PROGRAM P_Composite
VAR
	machine01				: Machine;
END_VAR

machine01.logStatus();

END_PROGRAM

(* stored: Version 1.1.0.1, ProductVersion 3.1.4024.12
   POU P_Composite: Id {42d147bc-3014-4419-b605-5661dbab23e6}, SpecialFunc None *)
